// Mitsubishi GX Works2 project: ghep dọc 1   PLC: FX1N/FX1NC

PROGRAM MAIN
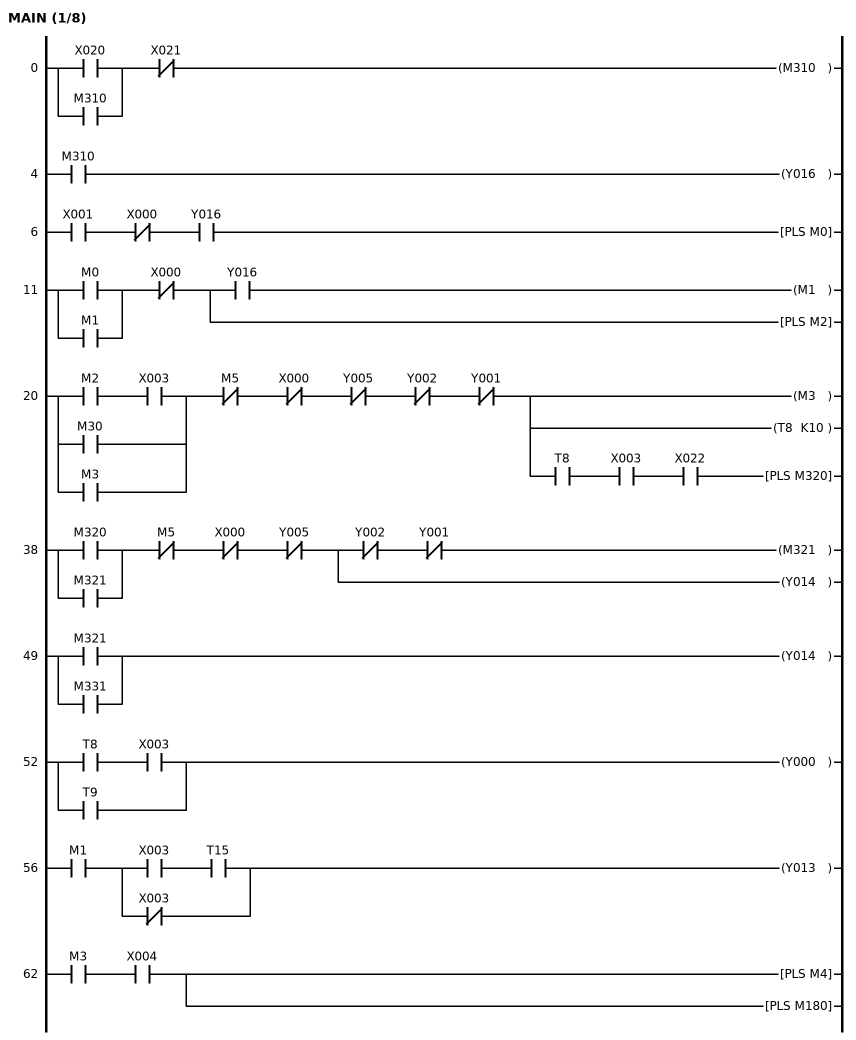
0     LD      X020
      OR      M310
      ANI     X021
      OUT     M310
4     LD      M310
      OUT     Y016
6     LD      X001
      ANI     X000
      AND     Y016
      PLS     M0
11    LD      M0
      OR      M1
      ANI     X000
      MPS
      AND     Y016
      OUT     M1
      MPP
      PLS     M2
20    LD      M2
      AND     X003
      OR      M30
      OR      M3
      ANI     M5
      ANI     X000
      ANI     Y005
      ANI     Y002
      ANI     Y001
      OUT     M3
      OUT     T8 K10
      AND     T8
      AND     X003
      AND     X022
      PLS     M320
38    LD      M320
      OR      M321
      ANI     M5
      ANI     X000
      ANI     Y005
      MPS
      ANI     Y002
      ANI     Y001
      OUT     M321
      MPP
      OUT     Y014
49    LD      M321
      OR      M331
      OUT     Y014
52    LD      T8
      AND     X003
      OR      T9
      OUT     Y000
56    LD      M1
      LD      X003
      AND     T15
      ORI     X003
      ANB
      OUT     Y013
62    LD      M3
      AND     X004
      PLS     M4
      PLS     M180
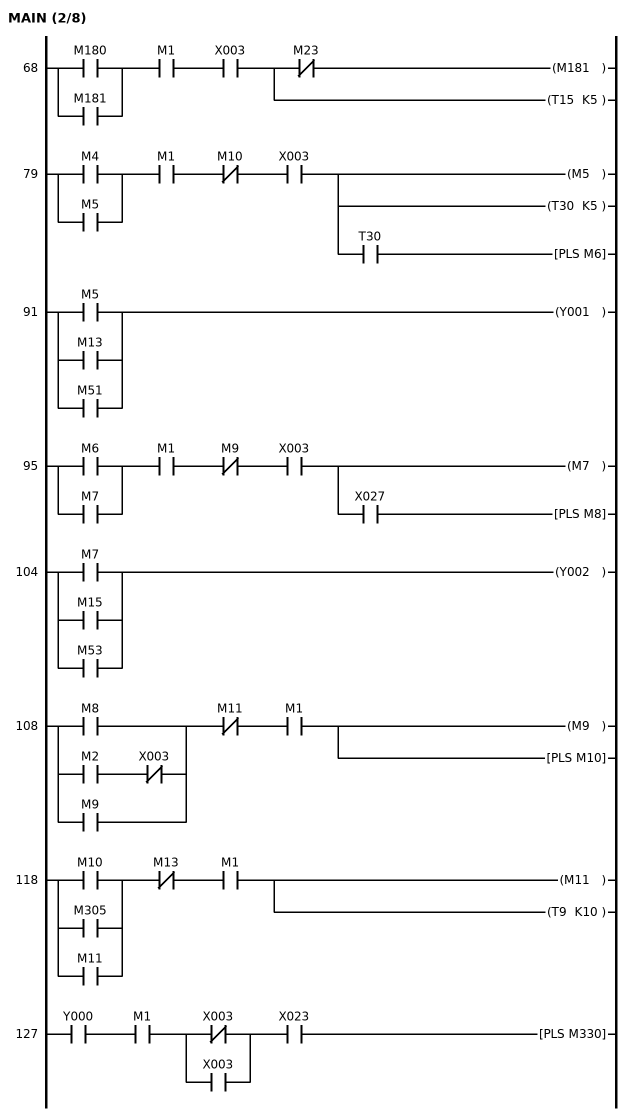
68    LD      M180
      OR      M181
      AND     M1
      AND     X003
      MPS
      ANI     M23
      OUT     M181
      MPP
      OUT     T15 K5
79    LD      M4
      OR      M5
      AND     M1
      ANI     M10
      AND     X003
      OUT     M5
      OUT     T30 K5
      AND     T30
      PLS     M6
91    LD      M5
      OR      M13
      OR      M51
      OUT     Y001
95    LD      M6
      OR      M7
      AND     M1
      ANI     M9
      AND     X003
      OUT     M7
      AND     X027
      PLS     M8
104   LD      M7
      OR      M15
      OR      M53
      OUT     Y002
108   LD      M8
      LD      M2
      ANI     X003
      ORB
      OR      M9
      ANI     M11
      AND     M1
      OUT     M9
      PLS     M10
118   LD      M10
      OR      M305
      OR      M11
      ANI     M13
      AND     M1
      OUT     M11
      OUT     T9 K10
127   LD      Y000
      AND     M1
      LDI     X003
      OR      X003
      ANB
      AND     X023
      PLS     M330
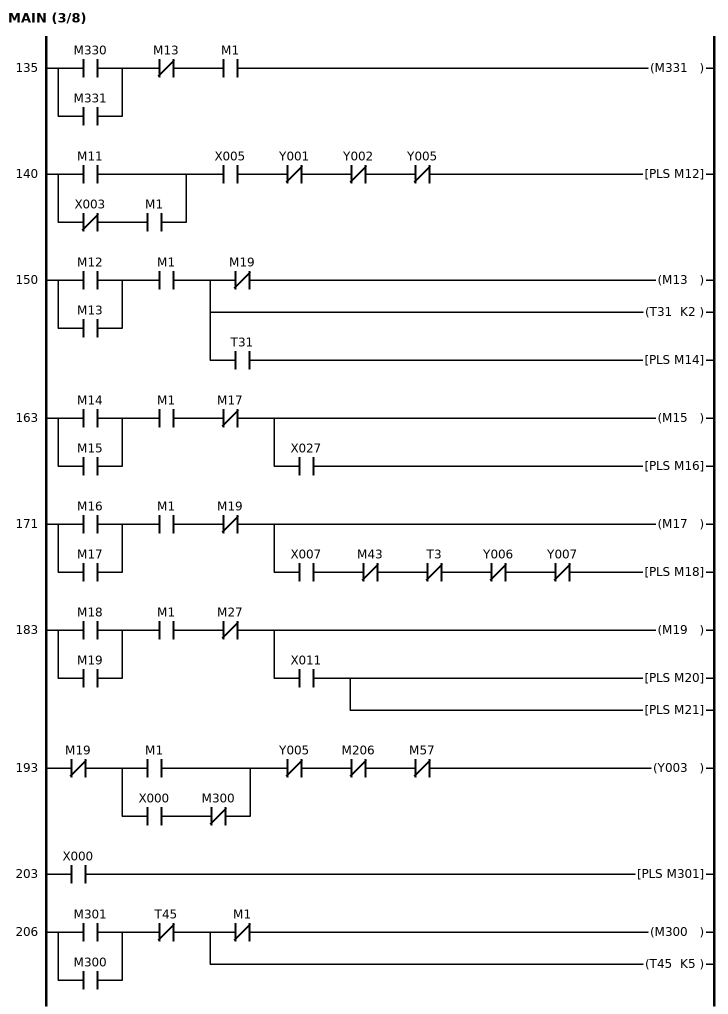
135   LD      M330
      OR      M331
      ANI     M13
      AND     M1
      OUT     M331
140   LD      M11
      LDI     X003
      AND     M1
      ORB
      AND     X005
      ANI     Y001
      ANI     Y002
      ANI     Y005
      PLS     M12
150   LD      M12
      OR      M13
      AND     M1
      MPS
      ANI     M19
      OUT     M13
      MPP
      OUT     T31 K2
      AND     T31
      PLS     M14
163   LD      M14
      OR      M15
      AND     M1
      ANI     M17
      OUT     M15
      AND     X027
      PLS     M16
171   LD      M16
      OR      M17
      AND     M1
      ANI     M19
      OUT     M17
      AND     X007
      ANI     M43
      ANI     T3
      ANI     Y006
      ANI     Y007
      PLS     M18
183   LD      M18
      OR      M19
      AND     M1
      ANI     M27
      OUT     M19
      AND     X011
      PLS     M20
      PLS     M21
193   LDI     M19
      LD      M1
      LD      X000
      ANI     M300
      ORB
      ANB
      ANI     Y005
      ANI     M206
      ANI     M57
      OUT     Y003
203   LD      X000
      PLS     M301
206   LD      M301
      OR      M300
      ANI     T45
      MPS
      ANI     M1
      OUT     M300
      MPP
      OUT     T45 K5
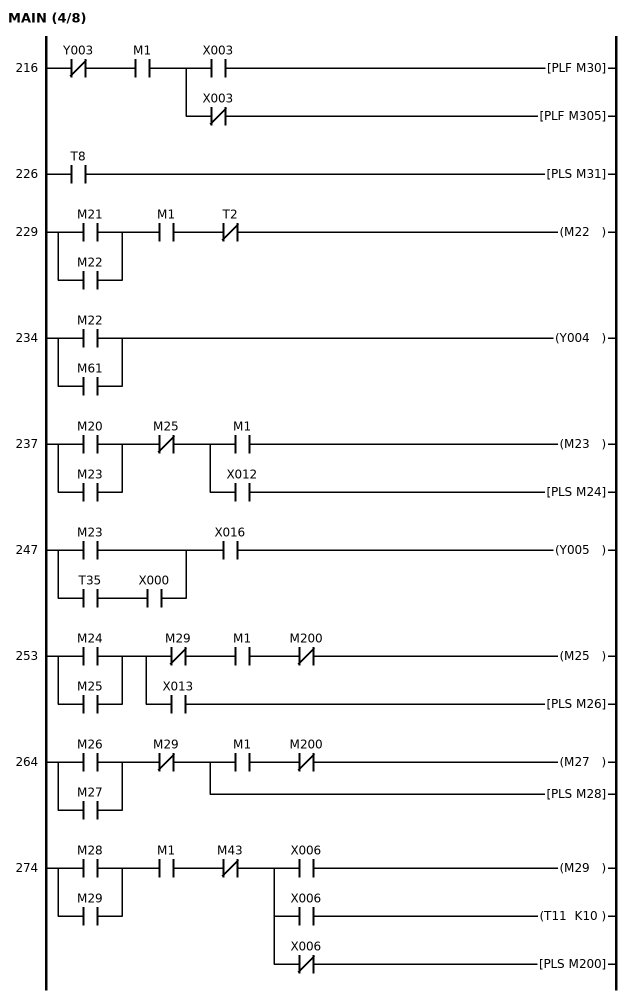
216   LDI     Y003
      AND     M1
      MPS
      AND     X003
      PLF     M30
      MPP
      ANI     X003
      PLF     M305
226   LD      T8
      PLS     M31
229   LD      M21
      OR      M22
      AND     M1
      ANI     T2
      OUT     M22
234   LD      M22
      OR      M61
      OUT     Y004
237   LD      M20
      OR      M23
      ANI     M25
      MPS
      AND     M1
      OUT     M23
      MPP
      AND     X012
      PLS     M24
247   LD      M23
      LD      T35
      AND     X000
      ORB
      AND     X016
      OUT     Y005
253   LD      M24
      OR      M25
      MPS
      ANI     M29
      AND     M1
      ANI     M200
      OUT     M25
      MPP
      AND     X013
      PLS     M26
264   LD      M26
      OR      M27
      ANI     M29
      MPS
      AND     M1
      ANI     M200
      OUT     M27
      MPP
      PLS     M28
274   LD      M28
      OR      M29
      AND     M1
      ANI     M43
      MPS
      AND     X006
      OUT     M29
      MRD
      AND     X006
      OUT     T11 K10
      MPP
      ANI     X006
      PLS     M200
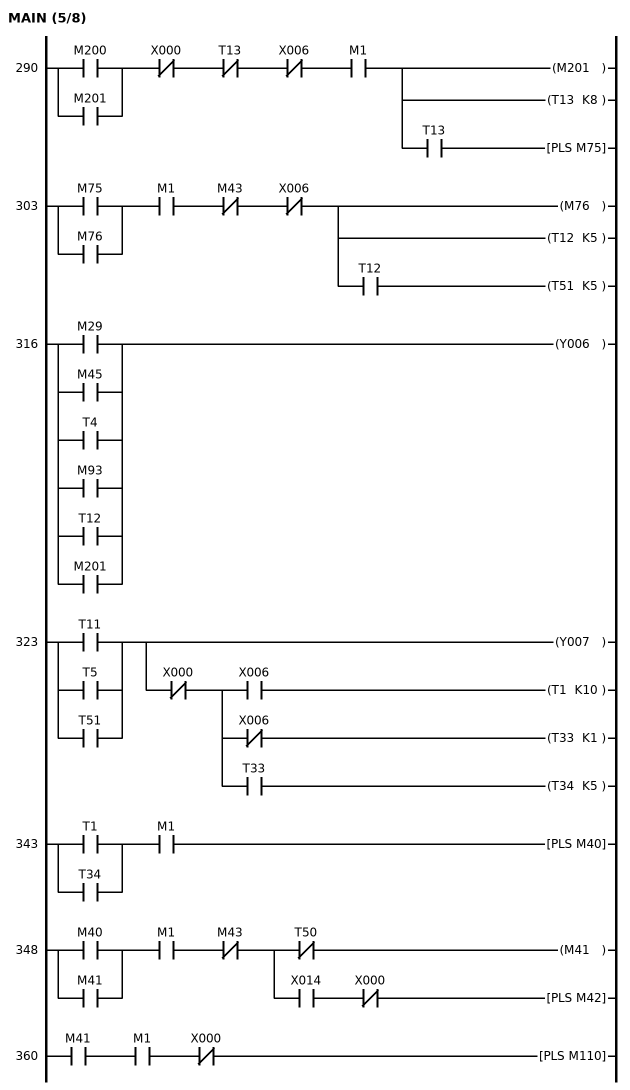
290   LD      M200
      OR      M201
      ANI     X000
      ANI     T13
      ANI     X006
      AND     M1
      OUT     M201
      OUT     T13 K8
      AND     T13
      PLS     M75
303   LD      M75
      OR      M76
      AND     M1
      ANI     M43
      ANI     X006
      OUT     M76
      OUT     T12 K5
      AND     T12
      OUT     T51 K5
316   LD      M29
      OR      M45
      OR      T4
      OR      M93
      OR      T12
      OR      M201
      OUT     Y006
323   LD      T11
      OR      T5
      OR      T51
      OUT     Y007
      ANI     X000
      MPS
      AND     X006
      OUT     T1 K10
      MRD
      ANI     X006
      OUT     T33 K1
      MPP
      AND     T33
      OUT     T34 K5
343   LD      T1
      OR      T34
      AND     M1
      PLS     M40
348   LD      M40
      OR      M41
      AND     M1
      ANI     M43
      MPS
      ANI     T50
      OUT     M41
      MPP
      AND     X014
      ANI     X000
      PLS     M42
360   LD      M41
      AND     M1
      ANI     X000
      PLS     M110
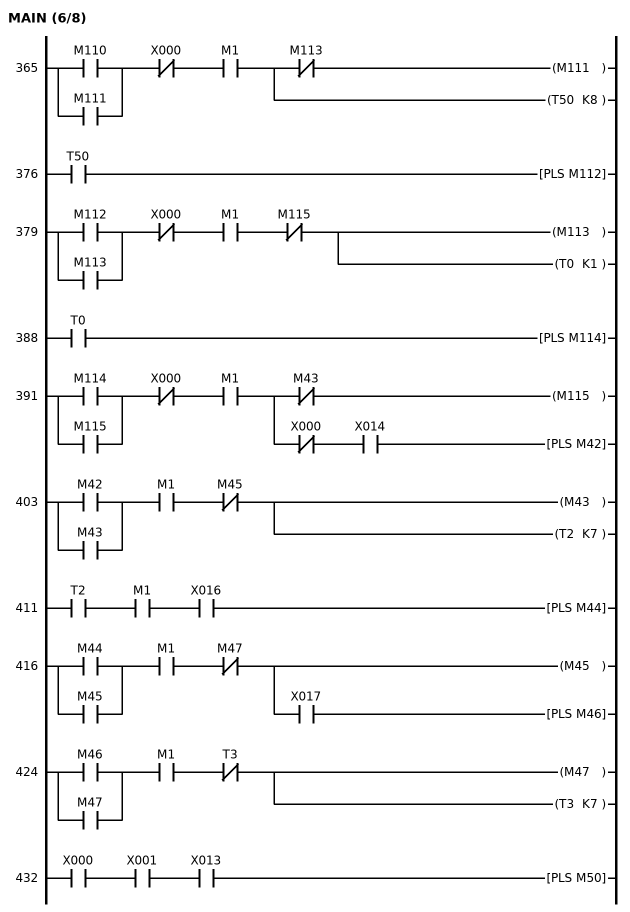
365   LD      M110
      OR      M111
      ANI     X000
      AND     M1
      MPS
      ANI     M113
      OUT     M111
      MPP
      OUT     T50 K8
376   LD      T50
      PLS     M112
379   LD      M112
      OR      M113
      ANI     X000
      AND     M1
      ANI     M115
      OUT     M113
      OUT     T0 K1
388   LD      T0
      PLS     M114
391   LD      M114
      OR      M115
      ANI     X000
      AND     M1
      MPS
      ANI     M43
      OUT     M115
      MPP
      ANI     X000
      AND     X014
      PLS     M42
403   LD      M42
      OR      M43
      AND     M1
      ANI     M45
      OUT     M43
      OUT     T2 K7
411   LD      T2
      AND     M1
      AND     X016
      PLS     M44
416   LD      M44
      OR      M45
      AND     M1
      ANI     M47
      OUT     M45
      AND     X017
      PLS     M46
424   LD      M46
      OR      M47
      AND     M1
      ANI     T3
      OUT     M47
      OUT     T3 K7
432   LD      X000
      AND     X001
      AND     X013
      PLS     M50
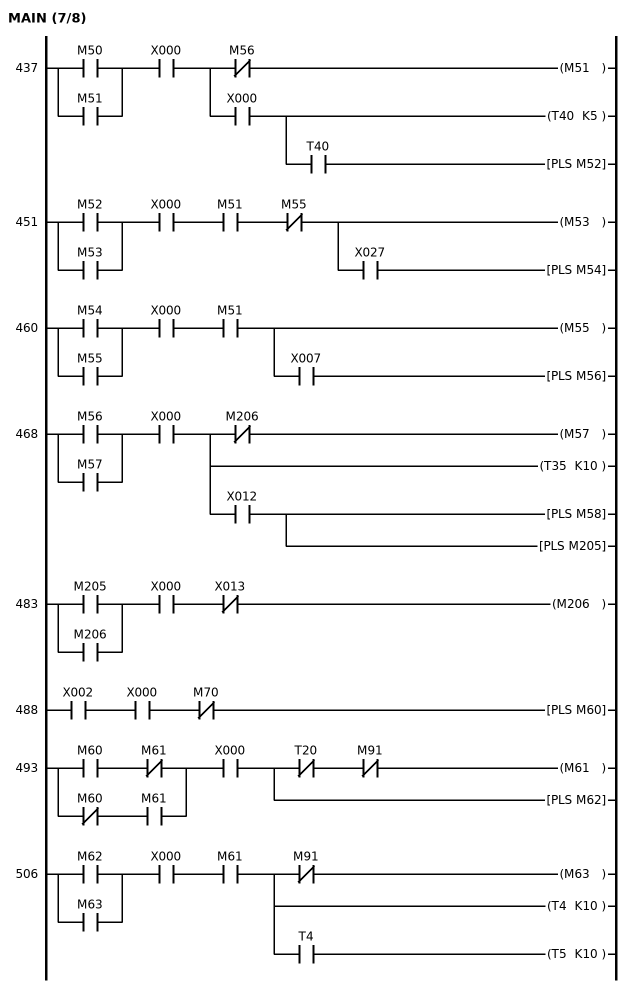
437   LD      M50
      OR      M51
      AND     X000
      MPS
      ANI     M56
      OUT     M51
      MPP
      AND     X000
      OUT     T40 K5
      AND     T40
      PLS     M52
451   LD      M52
      OR      M53
      AND     X000
      AND     M51
      ANI     M55
      OUT     M53
      AND     X027
      PLS     M54
460   LD      M54
      OR      M55
      AND     X000
      AND     M51
      OUT     M55
      AND     X007
      PLS     M56
468   LD      M56
      OR      M57
      AND     X000
      MPS
      ANI     M206
      OUT     M57
      MPP
      OUT     T35 K10
      AND     X012
      PLS     M58
      PLS     M205
483   LD      M205
      OR      M206
      AND     X000
      ANI     X013
      OUT     M206
488   LD      X002
      AND     X000
      ANI     M70
      PLS     M60
493   LD      M60
      ANI     M61
      LDI     M60
      AND     M61
      ORB
      AND     X000
      MPS
      ANI     T20
      ANI     M91
      OUT     M61
      MPP
      PLS     M62
506   LD      M62
      OR      M63
      AND     X000
      AND     M61
      MPS
      ANI     M91
      OUT     M63
      MPP
      OUT     T4 K10
      AND     T4
      OUT     T5 K10
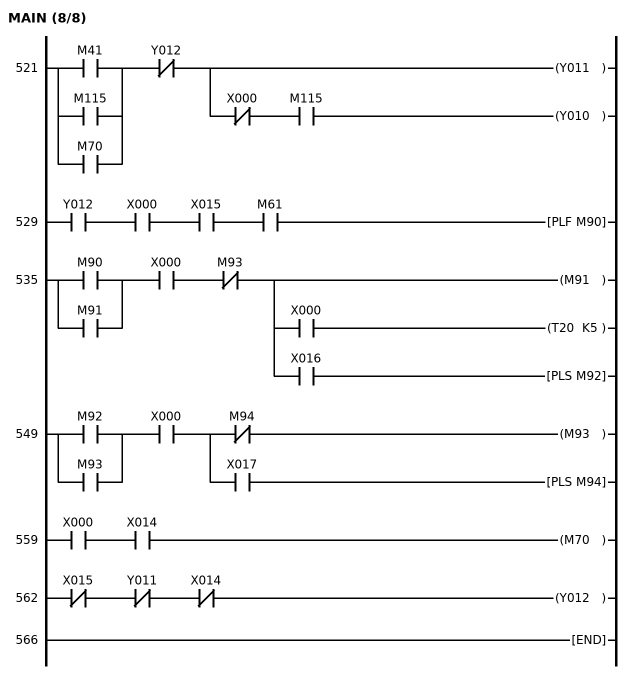
521   LD      M41
      OR      M115
      OR      M70
      ANI     Y012
      OUT     Y011
      ANI     X000
      AND     M115
      OUT     Y010
529   LD      Y012
      AND     X000
      AND     X015
      AND     M61
      PLF     M90
535   LD      M90
      OR      M91
      AND     X000
      ANI     M93
      OUT     M91
      MPS
      AND     X000
      OUT     T20 K5
      MPP
      AND     X016
      PLS     M92
549   LD      M92
      OR      M93
      AND     X000
      MPS
      ANI     M94
      OUT     M93
      MPP
      AND     X017
      PLS     M94
559   LD      X000
      AND     X014
      OUT     M70
562   LDI     X015
      ANI     Y011
      ANI     X014
      OUT     Y012
566   END
END_PROGRAM
